INTERFACE I_Axis

METHOD InPosition : BOOL
VAR_INPUT
END_VAR
END_METHOD

METHOD MoveAbsolute : BOOL
VAR_INPUT
	target : REAL;
END_VAR
END_METHOD

END_INTERFACE

(* stored: Version 1.1.0.1
   Itf I_Axis: Id {f04d6db4-ff92-4d67-b285-2162cf4a04b7}
   Method InPosition: Id {c6a586ca-1224-4e8d-98b7-7b51ddb11535}
   Method MoveAbsolute: Id {f2127f6f-c436-4cf6-ae87-0537fa73bb4e} *)
